# EPICS StreamDevice protocol: mc05/proto/encRead.proto
# Streams protocol file to supplement the pmacStreams protocol
# Created on 10/2015
# This file needs to be included after pmac proto, as it does not set serial communication parameters
# 0 suffix for VME, 1 suffix for GeoBrick - the only difference is an additional CR in "out"

# use "streamReload" to reload this file without restarting the IOC

ExtraInput = Ignore;
ReadTimeout = 500;
##OutTerminator = "";
InTerminator = ACK;
Separator = CR;

#out"M401" ENC4 24 bit counter position
getPos{ out"\$1" CR; in "%f";
}
